// TIA Portal V20 export
// export: Created 2025-12-01T14:57:14.8693678Z, ExportSetting None, DisplayName Totally Integrated Automation Portal, DisplayVersion V20 Update 3, DisplayName TIA Portal Openness, DisplayVersion V20 Update 3, DisplayName TIA Portal Version Control Interface, DisplayVersion V20 Update 3, DisplayName STEP 7 Professional, DisplayVersion V20 Update 3, DisplayName STEP 7 Safety, DisplayVersion V20 Update 2, DisplayName WinCC Basic/Comfort/Advanced, DisplayVersion V20 Update 3, DisplayName WinCC Professional, DisplayVersion V20 Update 3, DisplayName WinCC Unified, DisplayVersion V20 Update 3
FUNCTION_BLOCK "FB830_PasarDatosEntrePLCs_Origen"   // FB830, LAD
{ S7_Optimized_Access := 'FALSE' }
// stored: AutoNumber false, SetENOAutomatically false
   VAR_INPUT
      Mesa : UInt;
      OrdenEvacuar : Bool;
      In_BorrarUT : Bool;
   END_VAR
   VAR_OUTPUT
      Out_Mckey_01 : "UDT_EntrePLCs";
      Out_McKey_02 : "UDT_EntrePLCs";
      Out_DatosUT : Bool;
      OrdenEvacuar_OK : Bool;
   END_VAR
   VAR
      MMckeyUT_01 : "UDT_EntrePLCs";
      MMcKeyUT_02 : "UDT_EntrePLCs";
      NumeroUT_01 { ExternalAccessible := 'False'; ExternalVisible := 'False'; ExternalWritable := 'False'} : UInt;
      NumeroUT_02 { ExternalAccessible := 'False'; ExternalVisible := 'False'; ExternalWritable := 'False'} : UInt;
      ExisteUT_01 : Bool;
      ExisteUT_02 : Bool;
      MFP_BorrarUT : Bool;
      MDatosUT : Bool;
      MOrdenOK : Bool;
   END_VAR
   VAR_TEMP
      EstadoZona : "EstadoZona";
      EstadoVI : "EstadosMesa";
      Mckey_01 : "UDT_EntrePLCs";
      Mckey_02 : "UDT_EntrePLCs";
      P_Temporal : DWord;
      ValorReturn : Int;
      Cero : Byte;
      OrdenBorrarUT : Bool;
   END_VAR
   VAR_TEMP   // added for the SCL form of the ladder/FBD networks
      _w1 : Bool;
      _w2 : Bool;
      _w3 : Bool;
   END_VAR
BEGIN

REGION Network 1: Inicializar Variables
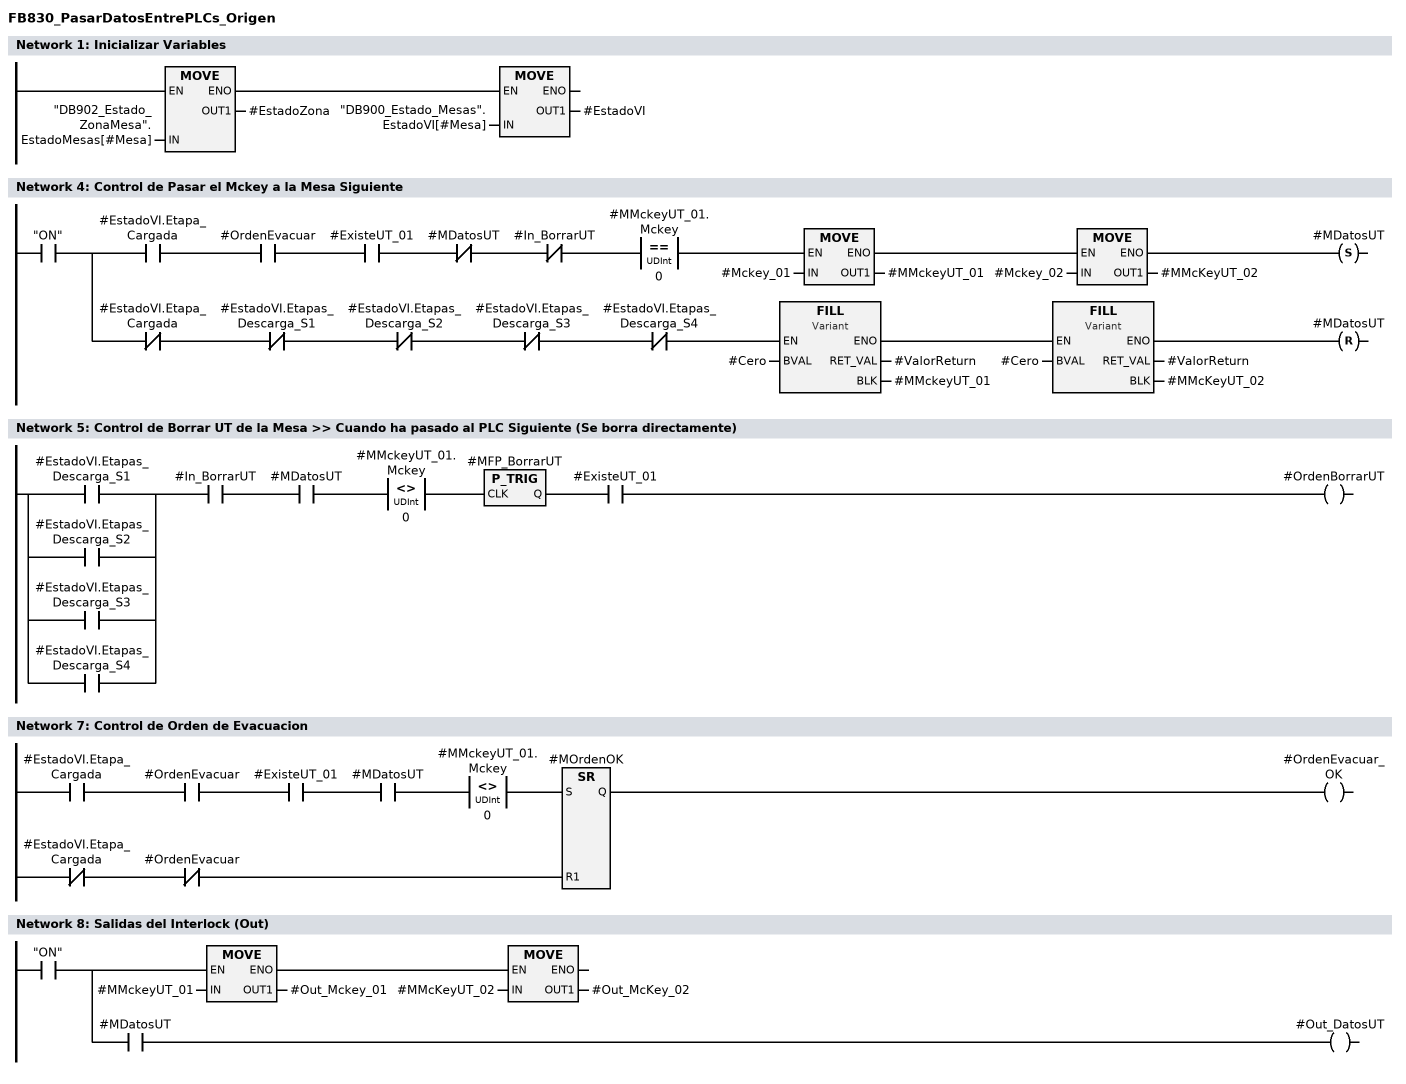
   RUNG wire#powerrail
      Move(in := "DB902_Estado_ZonaMesa".EstadoMesas[#Mesa], out1 => #EstadoZona)
      Move(in := "DB900_Estado_Mesas".EstadoVI[#Mesa], out1 => #EstadoVI)
   END_RUNG
   // the same network as SCL:
   #EstadoZona := "DB902_Estado_ZonaMesa".EstadoMesas[#Mesa];
   #EstadoVI := "DB900_Estado_Mesas".EstadoVI[#Mesa];
END_REGION

NETWORK
TITLE = ---
/////////////////////////////////////////////////////////////////////////////////
/////////////////////////////////////////////////////////////////////////////////
/////////////////////////////////////////////////////////////////////////////////
/// --- Inicializar Variables
      L     0;
      T     #Cero;


NETWORK
TITLE = Obtener Datos UT en la Mesa Actual
/////////////////////////////////////////////////////////////////////////////////
/////////////////////////////////////////////////////////////////////////////////
/////////////////////////////////////////////////////////////////////////////////
/// --- Inicializar

      SET;  // Inicializacion
      R     #ExisteUT_01;  // No Existe UT
      R     #ExisteUT_02;

      L     0;
      T     #NumeroUT_01;
      T     #NumeroUT_02;

      CALL  FILL
      ( BVAL    := #Cero,
        RET_VAL := #ValorReturn,
        BLK     := #Mckey_01
      );
      CALL  FILL
      ( BVAL    := #Cero,
        RET_VAL := #ValorReturn,
        BLK     := #Mckey_02
      );


/////////////////////////////////////////////////////////////////////////////////
/// --- Buscar Primera UT de la Mesa

      L     "DB810_ColasMesas".Colas[#Mesa].UT_PrimeraMesa;
      T     #NumeroUT_01;

      L     #NumeroUT_01;  // No hay UT's ?
      L     0;
      ==I;
      JC    FinDatosUTs_EnMesa;


/////////////////////////////////////////////////////////////////////////////////
/////////////////////////////////////////////////////////////////////////////////
/////////////////////////////////////////////////////////////////////////////////
/// --- Existe UT en la Mesa >>> Recoger Datos
      SET;
      S     #ExisteUT_01;  // Existe UT

      L     "DB812_UTs_Control".UT[#NumeroUT_01].Mckey;
      T     #Mckey_01.Mckey;
      L     "DB812_UTs_Control".UT[#NumeroUT_01].Grupo;
      T     #Mckey_01.Grupo;
      L     "DB812_UTs_Control".UT[#NumeroUT_01].TipoCarga;
      T     #Mckey_01.TipoCarga;

      L     "DB812_UTs_Control".UT[#NumeroUT_01].MesaDestino;
      T     #Mckey_01.MesaDestino;
      L     "DB813_UTs_Ruta".UT[#NumeroUT_01].Ruta[0];
      T     #Mckey_01.MesaSiguienteRuta;

      SET;
      A     "DB812_UTs_Control".UT[#NumeroUT_01].AtributosDelaCarga.Vacia;
      =     #Mckey_01.AtributosDelaCarga.Vacia;
      SET;
      A     "DB812_UTs_Control".UT[#NumeroUT_01].AtributosDelaCarga.Pila;
      =     #Mckey_01.AtributosDelaCarga.Pila;
      SET;
      A     "DB812_UTs_Control".UT[#NumeroUT_01].AtributosDelaCarga.Remontada;
      =     #Mckey_01.AtributosDelaCarga.Remontada;


/////////////////////////////////////////////////////////////////////////////////
/// --- Comprobar si puede haber mas

      L     "DB812_UTs_Control".UT[#NumeroUT_01].Grupo;
      L     0;  // Si es Grupo = 0 No hay mas
      ==I;
      JC    FinDatosUTs_EnMesa;

      L     "DB812_UTs_Control".UT[#NumeroUT_01].UT_SiguienteMesa;  // Hay mas UTs en la Mesa
      L     0;
      ==I;
      JC    FinDatosUTs_EnMesa;


/////////////////////////////////////////////////////////////////////////////////
/////////////////////////////////////////////////////////////////////////////////
/////////////////////////////////////////////////////////////////////////////////
/// --- Recoger datos de la Segunda UT

      L     "DB812_UTs_Control".UT[#NumeroUT_01].UT_SiguienteMesa;
      T     #NumeroUT_02;  // Puntero a los Datos de la UT

      SET;
      S     #ExisteUT_02;  // Existe UT

      L     "DB812_UTs_Control".UT[#NumeroUT_02].Mckey;
      T     #Mckey_02.Mckey;
      L     "DB812_UTs_Control".UT[#NumeroUT_02].Grupo;
      T     #Mckey_02.Grupo;
      L     "DB812_UTs_Control".UT[#NumeroUT_02].TipoCarga;
      T     #Mckey_02.TipoCarga;

      L     "DB812_UTs_Control".UT[#NumeroUT_02].MesaDestino;
      T     #Mckey_02.MesaDestino;
      L     "DB813_UTs_Ruta".UT[#NumeroUT_02].Ruta[0];
      T     #Mckey_02.MesaSiguienteRuta;

      SET;
      A     "DB812_UTs_Control".UT[#NumeroUT_02].AtributosDelaCarga.Vacia;
      =     #Mckey_02.AtributosDelaCarga.Vacia;
      SET;
      A     "DB812_UTs_Control".UT[#NumeroUT_02].AtributosDelaCarga.Pila;
      =     #Mckey_02.AtributosDelaCarga.Pila;
      SET;
      A     "DB812_UTs_Control".UT[#NumeroUT_02].AtributosDelaCarga.Remontada;
      =     #Mckey_02.AtributosDelaCarga.Remontada;


/////////////////////////////////////////////////////////////////////////////////
/// --- Comprobar si son pareja

      L     "DB812_UTs_Control".UT[#NumeroUT_01].Grupo;  // Son el mismo Grupo
      L     "DB812_UTs_Control".UT[#NumeroUT_02].Grupo;
      ==I;
      JC    FinDatosUTs_EnMesa;


/////////////////////////////////////////////////////////////////////////////////
/// --- Borrado de Datos no son el mismo grupo

      SET;
      R     #ExisteUT_02;

      L     0;
      T     #NumeroUT_02;

      CALL  FILL
      ( BVAL    := #Cero,
        RET_VAL := #ValorReturn,
        BLK     := #Mckey_01
      );


/////////////////////////////////////////////////////////////////////////////////
/////////////////////////////////////////////////////////////////////////////////
/////////////////////////////////////////////////////////////////////////////////
/// --- Final de Lectura de Datos de la UT en La Mesa
FinDatosUTs_EnMesa:NOP   0;



REGION Network 4: Control de Pasar el Mckey a la Mesa Siguiente
   RUNG wire#powerrail
      Contact( "ON" )
      wire#w1
      Contact( #EstadoVI.Etapa_Cargada )
      Contact( #OrdenEvacuar )
      Contact( #ExisteUT_01 )
      I_Contact( #MDatosUT )
      I_Contact( #In_BorrarUT )
      { S7_Templates := "SrcType := UDInt" } EQ_Contact(in1 := #MMckeyUT_01.Mckey, in2 := 0)
      { S7_GenerateENO := "TRUE" } Move(in := #Mckey_01, out1 => #MMckeyUT_01)
      { S7_GenerateENO := "TRUE" } Move(in := #Mckey_02, out1 => #MMcKeyUT_02)
      S_Coil( #MDatosUT )
   END_RUNG
   RUNG wire#w1
      I_Contact( #EstadoVI.Etapa_Cargada )
      I_Contact( #EstadoVI.Etapas_Descarga_S1 )
      I_Contact( #EstadoVI.Etapas_Descarga_S2 )
      I_Contact( #EstadoVI.Etapas_Descarga_S3 )
      I_Contact( #EstadoVI.Etapas_Descarga_S4 )
      { S7_Templates := "ptr_type := Variant" } FILL(BVAL := #Cero, RET_VAL => #ValorReturn, BLK => #MMckeyUT_01)
      { S7_Templates := "ptr_type := Variant" } FILL(BVAL := #Cero, RET_VAL => #ValorReturn, BLK => #MMcKeyUT_02)
      R_Coil( #MDatosUT )
   END_RUNG
   // the same network as SCL:
   // ENO of a box is taken as its EN; it also drops when the box reports an error
   #_w1 := "ON" AND #EstadoVI.Etapa_Cargada AND #OrdenEvacuar AND #ExisteUT_01 AND NOT #MDatosUT AND NOT #In_BorrarUT AND (#MMckeyUT_01.Mckey = 0);
   IF #_w1 THEN
       #MMckeyUT_01 := #Mckey_01;
       #MMcKeyUT_02 := #Mckey_02;
       #MDatosUT := TRUE;
   END_IF;
   #ValorReturn := FILL(EN := "ON" AND NOT #EstadoVI.Etapa_Cargada AND NOT #EstadoVI.Etapas_Descarga_S1 AND NOT #EstadoVI.Etapas_Descarga_S2 AND NOT #EstadoVI.Etapas_Descarga_S3 AND NOT #EstadoVI.Etapas_Descarga_S4,
                        BVAL := #Cero,
                        BLK => #MMckeyUT_01,
                        ENO => #_w2);
   #ValorReturn := FILL(EN := #_w2, BVAL := #Cero, BLK => #MMcKeyUT_02, ENO => #_w3);
   IF #_w3 THEN #MDatosUT := FALSE; END_IF;
END_REGION

REGION Network 5: Control de Borrar UT de la Mesa >> Cuando ha pasado al PLC Siguiente (Se borra directamente)
   RUNG wire#powerrail
      Contact( #EstadoVI.Etapas_Descarga_S1 )
      wire#w1
      Contact( #In_BorrarUT )
      Contact( #MDatosUT )
      { S7_Templates := "SrcType := UDInt" } NE_Contact(in1 := #MMckeyUT_01.Mckey, in2 := 0)
      P_Trig( #MFP_BorrarUT )
      Contact( #ExisteUT_01 )
      Coil( #OrdenBorrarUT )
   END_RUNG
   RUNG wire#powerrail
      Contact( #EstadoVI.Etapas_Descarga_S2 )
   END_RUNG wire#w1
   RUNG wire#powerrail
      Contact( #EstadoVI.Etapas_Descarga_S3 )
   END_RUNG wire#w1
   RUNG wire#powerrail
      Contact( #EstadoVI.Etapas_Descarga_S4 )
   END_RUNG wire#w1
   // the same network as SCL:
   #_w1 := (#EstadoVI.Etapas_Descarga_S1 OR #EstadoVI.Etapas_Descarga_S2 OR #EstadoVI.Etapas_Descarga_S3 OR #EstadoVI.Etapas_Descarga_S4) AND #In_BorrarUT AND #MDatosUT AND (#MMckeyUT_01.Mckey <> 0);
   #_w2 := #_w1 AND NOT #MFP_BorrarUT;   // rising edge
   #MFP_BorrarUT := #_w1;
   #OrdenBorrarUT := #_w2 AND #ExisteUT_01;
END_REGION

NETWORK
TITLE = --
/////////////////////////////////////////////////////////////////////////////////
/////////////////////////////////////////////////////////////////////////////////
/////////////////////////////////////////////////////////////////////////////////
/// - Ordem de Borrar

      SET;  // Hay que BorrarUT
      AN    #OrdenBorrarUT;
      JC    FinBorrarUT_EnMesa;


/////////////////////////////////////////////////////////////////////////////////
/////////////////////////////////////////////////////////////////////////////////
/////////////////////////////////////////////////////////////////////////////////
      SET;  // Eliminar datos Memorizados
      R     #MDatosUT;

      CALL  FILL
      ( BVAL    := #Cero,
        RET_VAL := #ValorReturn,
        BLK     := #MMckeyUT_01
      );
      CALL  FILL
      ( BVAL    := #Cero,
        RET_VAL := #ValorReturn,
        BLK     := #MMcKeyUT_02
      );


/////////////////////////////////////////////////////////////////////////////////
      SET;
      AN    #ExisteUT_01;  // Existe UT 01 en la Mesa
      JC    FinBorrarUT_EnMesa;

      CALL  "FC722_EliminarUT_DeMesa"
      ( NumeroUT := #NumeroUT_01
      );  //Eliminar la Primera UT de la mesa


      AN    #ExisteUT_02;  // Existe UT 02 en la Mesa
      JC    FinBorrarUT_EnMesa;

      CALL  "FC722_EliminarUT_DeMesa"
      ( NumeroUT := #NumeroUT_02
      );  //Eliminar la Segunda UT de la mesa


/////////////////////////////////////////////////////////////////////////////////
/////////////////////////////////////////////////////////////////////////////////
/////////////////////////////////////////////////////////////////////////////////
FinBorrarUT_EnMesa:NOP   0;



REGION Network 7: Control de Orden de Evacuacion
   RUNG wire#powerrail
      Contact( #EstadoVI.Etapa_Cargada )
      Contact( #OrdenEvacuar )
      Contact( #ExisteUT_01 )
      Contact( #MDatosUT )
      { S7_Templates := "SrcType := UDInt" } NE_Contact(in1 := #MMckeyUT_01.Mckey, in2 := 0)
      S_SR(operand := #MOrdenOK, r1 := wire#w1)
      Coil( #OrdenEvacuar_OK )
   END_RUNG
   RUNG wire#powerrail
      I_Contact( #EstadoVI.Etapa_Cargada )
      I_Contact( #OrdenEvacuar )
   END_RUNG wire#w1
   // the same network as SCL:
   IF #EstadoVI.Etapa_Cargada AND #OrdenEvacuar AND #ExisteUT_01 AND #MDatosUT AND (#MMckeyUT_01.Mckey <> 0) THEN
       #MOrdenOK := TRUE;   // SR flip-flop
   END_IF;
   IF NOT #EstadoVI.Etapa_Cargada AND NOT #OrdenEvacuar THEN #MOrdenOK := FALSE; END_IF;
   #OrdenEvacuar_OK := #MOrdenOK;
END_REGION

REGION Network 8: Salidas del Interlock (Out)
   RUNG wire#powerrail
      Contact( "ON" )
      wire#w1
      Move(in := #MMckeyUT_01, out1 => #Out_Mckey_01)
      Move(in := #MMcKeyUT_02, out1 => #Out_McKey_02)
   END_RUNG
   RUNG wire#w1
      Contact( #MDatosUT )
      Coil( #Out_DatosUT )
   END_RUNG
   // the same network as SCL:
   IF "ON" THEN
       #Out_Mckey_01 := #MMckeyUT_01;
       #Out_McKey_02 := #MMcKeyUT_02;
   END_IF;
   #Out_DatosUT := "ON" AND #MDatosUT;
END_REGION
END_FUNCTION_BLOCK
